TEXTLIST Equipment_Status
  0 = 'ALARM'
  1 = 'HEALTHY'
   = ''
END_TEXTLIST

(* stored: Version 1.1.0.1, ProductVersion 3.1.4024.12
   TextList Equipment_Status: Id {a3412d9d-4b22-46be-b8c4-de583f02bfd1} *)
